(* CoDeSys 2.3 export: GETMODBUSREGISTERS.EXP *)

(* POU Modbus/getModbusRegisters, ST *)
FUNCTION getModbusRegisters : BOOL
VAR_INPUT
END_VAR
VAR
END_VAR
K14UZSPumpSpeed := WORD_TO_USINT(MB_W_01);
END_FUNCTION
